// TIA Portal V16 export
// export: Created 2022-09-05T21:51:21.0234373Z, ExportSetting WithDefaults, DisplayName Totally Integrated Automation Portal, DisplayVersion V16, DisplayName TIA Portal Version Control Interface, DisplayVersion V16, DisplayName TIA Portal Openness, DisplayVersion V16, DisplayName SINAMICS Startdrive Advanced, DisplayVersion V16, DisplayName SINAMICS Startdrive G130, G150, S120, S150, SINAMICS MV, S210, DisplayVersion V16, DisplayName SINAMICS Startdrive G110M, G120, G120C, G120D, G120P, DisplayVersion V16, DisplayName STEP 7 Professional, DisplayVersion V16, DisplayName STEP 7 Safety, DisplayVersion V16, DisplayName WinCC Professional, DisplayVersion V16
ORGANIZATION_BLOCK "Counter_Project"   // OB1, LAD, ProgramCycle
TITLE = "Main Program Sweep (Cycle)"
{ S7_Optimized_Access := 'TRUE' }
VERSION : 0.1
// stored: AutoNumber true, IsIECCheckEnabled false, SetENOAutomatically false
   VAR_INPUT
      Initial_Call : Bool;   // Initial call of this OB
      Remanence : Bool;   // =True, if remanent data are available
   END_VAR
BEGIN

REGION Network 1
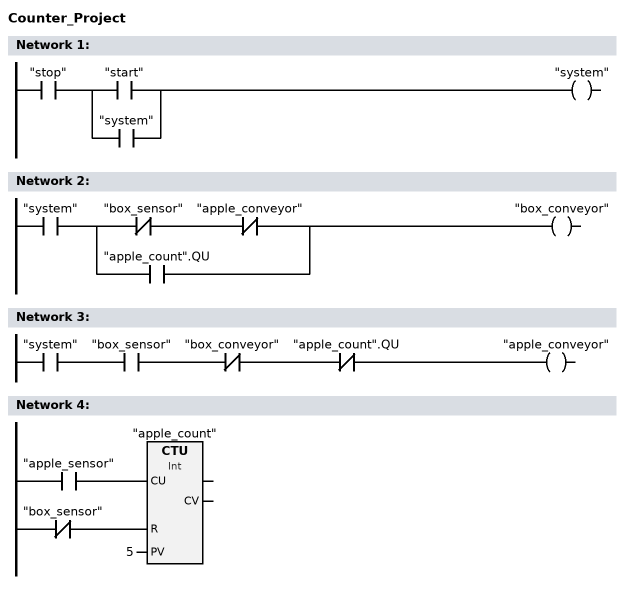
   RUNG wire#powerrail
      Contact( "stop" )
      wire#w1
      Contact( "start" )
      wire#w2
      Coil( "system" )
   END_RUNG
   RUNG wire#w1
      Contact( "system" )
   END_RUNG wire#w2
   // the same network as SCL:
   "system" := "stop" AND ("start" OR "system");
END_REGION

REGION Network 2
   RUNG wire#powerrail
      Contact( "system" )
      wire#w1
      I_Contact( "box_sensor" )
      I_Contact( "apple_conveyor" )
      wire#w2
      Coil( "box_conveyor" )
   END_RUNG
   RUNG wire#w1
      Contact( "apple_count".QU )
   END_RUNG wire#w2
   // the same network as SCL:
   "box_conveyor" := "system" AND ((NOT "box_sensor" AND NOT "apple_conveyor") OR "apple_count".QU);
END_REGION

REGION Network 3
   RUNG wire#powerrail
      Contact( "system" )
      Contact( "box_sensor" )
      I_Contact( "box_conveyor" )
      I_Contact( "apple_count".QU )
      Coil( "apple_conveyor" )
   END_RUNG
   // the same network as SCL:
   "apple_conveyor" := "system" AND "box_sensor" AND NOT "box_conveyor" AND NOT "apple_count".QU;
END_REGION

REGION Network 4
   RUNG wire#powerrail
      Contact( "apple_sensor" )
      { S7_Templates := "value_type := Int" } "apple_count".CTU(r := wire#w1, pv := 5, cv =>)
   END_RUNG
   RUNG wire#powerrail
      I_Contact( "box_sensor" )
   END_RUNG wire#w1
   // the same network as SCL:
   "apple_count".CTU(CU := "apple_sensor", R := NOT "box_sensor", PV := 5);
END_REGION
END_ORGANIZATION_BLOCK
